Universal Robots PolyScope program: palety_venclovsky.urp

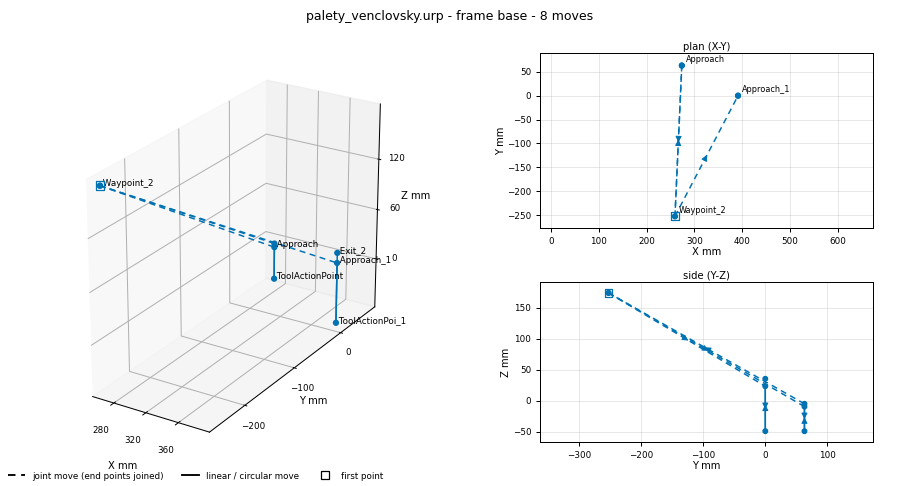
[picture p0: tool path of palety_venclovsky.urp in frame base, 8 of 8 moves have a stored position in this frame; points joined in program order, loops and branches not executed]
Program palety_venclovsky (installation=default directory=/programs/usbdisk createdIn=5.21.2 lastSavedIn=5.21.2 robotSerialNumber=20185300578)
Calibrated DH parameters: a=[-0.000189, -0.243548, -0.212949, 0.000139, -0.000171, 0]; d=[0.151928, 2.340352, -3.79233, 1.582506, 0.085299, 0.092103]; alpha=[1.570802, 0.003282, -0.008312, 1.570809, -1.571939, 0]; deltaTheta=[0, 0.031526, 6.30827, -0.05661, 0, 0]
InitVariablesNode variables(variable(name=Pallet_1_cnt, expression=1), variable(name=Pallet_1_lct, expression=1), variable(name=Pallet_1_lno, expression=1), variable(name=Pallet_1_sep, expression=False), variable(name=Pallet_1_tct, expression=1), variable(name=Pallet_2_cnt, expression=1), variable(name=Pallet_2_lct, expression=1), variable(name=Pallet_2_lno, expression=1), variable(name=Pallet_2_sep, expression=False), variable(name=Pallet_2_tct, expression=1), variable(name=qNearApproach, expression=[0,0,0,0,0,0]), variable(name=qNearApproach_1, expression=[0,0,0,0,0,0]))
BeforeStart
  pocitadlo := 0
  URCap Gripper Activate (Robotiq_Grippers, Robotiq Inc.) dataModel(ResetAndActivateKey=false)
Robot Program (runOnlyOnce=false)
  Call pas_on
  Wait DigitalInput pin=digital_in[2]; digitalValue=1
  URCap Gripper (Robotiq_Grippers, Robotiq Inc.) dataModel(position=100.0, force=54.0, speed=70.0, positionInDouble=100.0, forceInDouble=54.0, speedInDouble=70.0, slaveIds=[9], blocking=true, robotCompliant=false)
  MoveJ speed 60 deg/s, acceleration 80 deg/s^2 (useActiveTCP=true optimoveEnabled=false optiMoveSpeed=0.3 optiMoveAcceleration=0.09) feature=Base
    Waypoint Waypoint_2: TCP in base x=259.302 y=-252.628 z=173.963 mm, rx=-2.2194 ry=2.2233 rz=0.0001 rad; joints [-23.019, -99.618, -73.74, -96.577, 89.565, -23.023] deg; TCP offset x=0 y=0 z=150 mm, rx=0 ry=0 rz=0 rad
  Call pas_off
  If pocitadlo<6
    MoveL speed 180 mm/s, acceleration 1200 mm/s^2 (useActiveTCP=true optimoveEnabled=false optiMoveSpeed=0.3 optiMoveAcceleration=0.09) feature=Base
      MoveDirectionNode (selectedDirection=ZMinus)
        Until TOOL_CONTACT_DETECTION (allowActions=true retraction=0.005 decelerationAcceleration=3 decelerationAngularAcceleration=34.906585)
          MoveDirectionNode (selectedDirection=ZPlus)
            Until DISTANCE (allowActions=false deceleration=3 distanceNodeType=STOP) Distance=0.01; motionParameters(blendRadius=0)
          URCap Gripper (Robotiq_Grippers, Robotiq Inc.) dataModel(position=0.0, force=1.1764705882352942, speed=80.0, positionInDouble=0.0, forceInDouble=1.1764705882352942, speedInDouble=80.0, slaveIds=[9], blocking=true, robotCompliant=false)
          MoveDirectionNode (selectedDirection=ZMinus)
            Until DISTANCE (allowActions=false deceleration=3 distanceNodeType=STOP) Distance=0.025; motionParameters(blendRadius=0)
          pocitadlo := pocitadlo+1
          URCap Gripper (Robotiq_Grippers, Robotiq Inc.) dataModel(position=44.31372549019608, force=39.0, speed=70.0, positionInDouble=44.31372549019608, forceInDouble=39.0, speedInDouble=70.0, slaveIds=[9], blocking=true, robotCompliant=false)
          MoveDirectionNode (selectedDirection=ZPlus)
            Until DISTANCE (allowActions=false deceleration=3 distanceNodeType=STOP) Distance=0.06; motionParameters(blendRadius=0)
          Call pas_off
          URCap Palletizing (polyscope-pallet-impl, Universal Robots) dataModel(palletFeature=Base, isPalletizing=true, rememberTraversal=false, Length(key=objectHeight value=0.03 unit=M), Variable(key=referencePoint, variable(featureName=referencePoint)), Variable(key=separatorPoint, variable(featureName=separatorPoint)), Variable(key=qNearApproach, variable(name=qNearApproach, initializeExpression=[0,0,0,0,0,0])), Variable(key=layerCountingVariable, variable(name=Pallet_1_lct, initializeExpression=1)), Variable(key=layerNumberVariable, variable(name=Pallet_1_lno, initializeExpression=1)), Variable(key=handleSeparatorVariable, variable(name=Pallet_1_sep, initializeExpression=False)), Variable(key=totalCountVariable, variable(name=Pallet_1_tct, initializeExpression=1)), Variable(key=name, variable(name=Pallet_1)), Variable(key=globalCountingVariable, variable(name=Pallet_1_cnt, initializeExpression=1))); state(isChildrenLocked=true)
            URCap Patterns (polyscope-pallet-impl, Universal Robots) state(isChildrenLocked=true)
              URCap Pattern (polyscope-pallet-impl, Universal Robots) dataModel(UUID=a1afcf7f-e893-493d-b622-6c9d734d3802, patternType=GRID, rows=3, columns=2, Variable(key=nameVariable, variable(name=Grid_Pattern_1))); state(isChildrenLocked=true)
                URCap Item (polyscope-pallet-impl, Universal Robots) dataModel(UUID=0f84a695-5284-41e9-b3d2-203e22c0e9f4, patternType=GRID, index=0, calibrationDeltaTheta=[-9.679944364821003E-8, 0.03152637960071048, 6.308270136326222, -0.05660981424064361, 2.1302738175549285E-7, -3.4337321612454286E-7], calibrationA=[-1.89170984734602E-4, -0.24354794633452972, -0.2129485167088614, 1.3892904611349137E-4, -1.7067015336856014E-4, 0.0], calibrationD=[0.15192760230984942, 2.3403518756598336, -3.792330157129607, 1.5825055280731988, 0.08529876240250026, 0.09210299655971649], calibrationAlpha=[1.5708023866418512, 0.0032819461853986743, -0.008311935193061136, 1.570808769909054, -1.5719389687286305, 0.0], calibrationJointChecksum=[-1323472732, -1322302140, 655890344, -1781272900, -1781497016, -1329631202], calibrationStatus=2, calibrationValidChecksum=true, baseToFeature=[0.0, 0.0, 0.0, 0.0, 0.0, 0.0], TCPOffset=[3.46987351703687E-4, -7.600627802391707E-4, 0.2251579720144376, 1.768906187287919E-5, 2.956695373762668E-5, -0.002830388265502223], JointPositions(key=jointpositions, JointPosition(key=[1], Angle(key=pos value=0.712932 unit=RAD)), JointPosition(key=[2], Angle(key=pos value=-1.536445 unit=RAD)), JointPosition(key=[3], Angle(key=pos value=-2.239352 unit=RAD)), JointPosition(key=[4], Angle(key=pos value=-0.935455 unit=RAD)), JointPosition(key=[5], Angle(key=pos value=1.563636 unit=RAD)), JointPosition(key=[6], Angle(key=pos value=-0.86287 unit=RAD))), Variable(key=variable, variable(name=CornerItem_1)))
                URCap Item (polyscope-pallet-impl, Universal Robots) dataModel(UUID=4917496b-efcc-468c-8b87-0b4eec043f87, patternType=GRID, index=1, calibrationDeltaTheta=[-9.679944364821003E-8, 0.03152637960071048, 6.308270136326222, -0.05660981424064361, 2.1302738175549285E-7, -3.4337321612454286E-7], calibrationA=[-1.89170984734602E-4, -0.24354794633452972, -0.2129485167088614, 1.3892904611349137E-4, -1.7067015336856014E-4, 0.0], calibrationD=[0.15192760230984942, 2.3403518756598336, -3.792330157129607, 1.5825055280731988, 0.08529876240250026, 0.09210299655971649], calibrationAlpha=[1.5708023866418512, 0.0032819461853986743, -0.008311935193061136, 1.570808769909054, -1.5719389687286305, 0.0], calibrationJointChecksum=[-1323472732, -1322302140, 655890344, -1781272900, -1781497016, -1329631202], calibrationStatus=2, calibrationValidChecksum=true, baseToFeature=[0.0, 0.0, 0.0, 0.0, 0.0, 0.0], TCPOffset=[3.3288055820729356E-4, -7.179712004344516E-4, 0.22518613724958014, -6.51308584616644E-5, -5.815327347860047E-5, -0.0026860162808949157], JointPositions(key=jointpositions, JointPosition(key=[1], Angle(key=pos value=0.493777 unit=RAD)), JointPosition(key=[2], Angle(key=pos value=-2.007679 unit=RAD)), JointPosition(key=[3], Angle(key=pos value=-1.645848 unit=RAD)), JointPosition(key=[4], Angle(key=pos value=-1.057707 unit=RAD)), JointPosition(key=[5], Angle(key=pos value=1.564628 unit=RAD)), JointPosition(key=[6], Angle(key=pos value=-1.087185 unit=RAD))), Variable(key=variable, variable(name=CornerItem_2)))
                URCap Item (polyscope-pallet-impl, Universal Robots) dataModel(UUID=17d65b1d-739d-439a-9630-1cad21d49f15, patternType=GRID, index=2, calibrationDeltaTheta=[-9.679944364821003E-8, 0.03152637960071048, 6.308270136326222, -0.05660981424064361, 2.1302738175549285E-7, -3.4337321612454286E-7], calibrationA=[-1.89170984734602E-4, -0.24354794633452972, -0.2129485167088614, 1.3892904611349137E-4, -1.7067015336856014E-4, 0.0], calibrationD=[0.15192760230984942, 2.3403518756598336, -3.792330157129607, 1.5825055280731988, 0.08529876240250026, 0.09210299655971649], calibrationAlpha=[1.5708023866418512, 0.0032819461853986743, -0.008311935193061136, 1.570808769909054, -1.5719389687286305, 0.0], calibrationJointChecksum=[-1323472732, -1322302140, 655890344, -1781272900, -1781497016, -1329631202], calibrationStatus=2, calibrationValidChecksum=true, baseToFeature=[0.0, 0.0, 0.0, 0.0, 0.0, 0.0], TCPOffset=[3.5344163164441333E-4, -7.52499091124919E-4, 0.2251565599680179, 4.465585933927923E-6, 3.067966499632582E-5, -0.0027840861433366514], JointPositions(key=jointpositions, JointPosition(key=[1], Angle(key=pos value=0.3406 unit=RAD)), JointPosition(key=[2], Angle(key=pos value=-1.990637 unit=RAD)), JointPosition(key=[3], Angle(key=pos value=-1.675639 unit=RAD)), JointPosition(key=[4], Angle(key=pos value=-1.044914 unit=RAD)), JointPosition(key=[5], Angle(key=pos value=1.564624 unit=RAD)), JointPosition(key=[6], Angle(key=pos value=-1.242929 unit=RAD))), Variable(key=variable, variable(name=CornerItem_3)))
                URCap Item (polyscope-pallet-impl, Universal Robots) dataModel(UUID=e23a75e9-c512-4699-9fb0-38c1f641661b, patternType=GRID, index=3, calibrationDeltaTheta=[-9.679944364821003E-8, 0.03152637960071048, 6.308270136326222, -0.05660981424064361, 2.1302738175549285E-7, -3.4337321612454286E-7], calibrationA=[-1.89170984734602E-4, -0.24354794633452972, -0.2129485167088614, 1.3892904611349137E-4, -1.7067015336856014E-4, 0.0], calibrationD=[0.15192760230984942, 2.3403518756598336, -3.792330157129607, 1.5825055280731988, 0.08529876240250026, 0.09210299655971649], calibrationAlpha=[1.5708023866418512, 0.0032819461853986743, -0.008311935193061136, 1.570808769909054, -1.5719389687286305, 0.0], calibrationJointChecksum=[-1323472732, -1322302140, 655890344, -1781272900, -1781497016, -1329631202], calibrationStatus=2, calibrationValidChecksum=true, baseToFeature=[0.0, 0.0, 0.0, 0.0, 0.0, 0.0], TCPOffset=[3.5491326159248215E-4, -7.352154795082138E-4, 0.22516187238070134, -5.903850028089745E-5, 3.090088451041777E-5, -0.0028011796468691915], JointPositions(key=jointpositions, JointPosition(key=[1], Angle(key=pos value=0.501609 unit=RAD)), JointPosition(key=[2], Angle(key=pos value=-1.50856 unit=RAD)), JointPosition(key=[3], Angle(key=pos value=-2.27851 unit=RAD)), JointPosition(key=[4], Angle(key=pos value=-0.924139 unit=RAD)), JointPosition(key=[5], Angle(key=pos value=1.563638 unit=RAD)), JointPosition(key=[6], Angle(key=pos value=-1.073597 unit=RAD))), Variable(key=variable, variable(name=CornerItem_4)))
            URCap Layers (polyscope-pallet-impl, Universal Robots) dataModel(selectedPatterns=[a1afcf7f-e893-493d-b622-6c9d734d3802], separators=[false])
            URCap At Each Item (polyscope-pallet-impl, Universal Robots) dataModel(selectedPattern=a1afcf7f-e893-493d-b622-6c9d734d3802, selectedPosition=0f84a695-5284-41e9-b3d2-203e22c0e9f4, Approach_calibrationDeltaTheta=[-9.679944364821003E-8, 0.03152637960071048, 6.308270136326222, -0.05660981424064361, 2.1302738175549285E-7, -3.4337321612454286E-7], Approach_calibrationA=[-1.89170984734602E-4, -0.24354794633452972, -0.2129485167088614, 1.3892904611349137E-4, -1.7067015336856014E-4, 0.0], Approach_calibrationD=[0.15192760230984942, 2.3403518756598336, -3.792330157129607, 1.5825055280731988, 0.08529876240250026, 0.09210299655971649], Approach_calibrationAlpha=[1.5708023866418512, 0.0032819461853986743, -0.008311935193061136, 1.570808769909054, -1.5719389687286305, 0.0], Approach_calibrationJointChecksum=[-1323472732, -1322302140, 655890344, -1781272900, -1781497016, -1329631202], Approach_calibrationStatus=2, Approach_calibrationValidChecksum=true, Approach_baseToFeature=[0.0, 0.0, 0.0, 0.0, 0.0, 0.0], Approach_TCPOffset=[3.426090968767226E-4, -7.410222825070811E-4, 0.2251722220319323, -3.696212188149479E-5, -1.49889783493022E-5, -0.0027893122367816064], Exit_calibrationDeltaTheta=[-9.679944364821003E-8, 0.03152637960071048, 6.308270136326222, -0.05660981424064361, 2.1302738175549285E-7, -3.4337321612454286E-7], Exit_calibrationA=[-1.89170984734602E-4, -0.24354794633452972, -0.2129485167088614, 1.3892904611349137E-4, -1.7067015336856014E-4, 0.0], Exit_calibrationD=[0.15192760230984942, 2.3403518756598336, -3.792330157129607, 1.5825055280731988, 0.08529876240250026, 0.09210299655971649], Exit_calibrationAlpha=[1.5708023866418512, 0.0032819461853986743, -0.008311935193061136, 1.570808769909054, -1.5719389687286305, 0.0], Exit_calibrationJointChecksum=[-1323472732, -1322302140, 655890344, -1781272900, -1781497016, -1329631202], Exit_calibrationStatus=2, Exit_calibrationValidChecksum=true, Exit_baseToFeature=[0.0, 0.0, 0.0, 0.0, 0.0, 0.0], Exit_TCPOffset=[3.534060554490903E-4, -7.328819302233058E-4, 0.22516274782089438, -5.956694931654154E-5, 2.1349790715159343E-5, -0.0027647185049195196], currentWizardState=LANDING, Pose(key=refBaseToFeature, Position(key=posePosition, Length(key=X value=0 unit=M), Length(key=Y value=0 unit=M), Length(key=Z value=0 unit=M)), Rotation(key=poseRotation, Angle(key=RX value=0 unit=RAD), Angle(key=RY value=0 unit=RAD), Angle(key=RZ value=0 unit=RAD))), Pose(key=refPose, Position(key=posePosition, Length(key=X value=0.273602 unit=M), Length(key=Y value=0.063177 unit=M), Length(key=Z value=-0.048894 unit=M)), Rotation(key=poseRotation, Angle(key=RX value=-3.14157 unit=RAD), Angle(key=RY value=-0.000044 unit=RAD), Angle(key=RZ value=0.000006 unit=RAD))), JointPositions(key=Approach_jointpositions, JointPosition(key=[1], Angle(key=pos value=0.712584 unit=RAD)), JointPosition(key=[2], Angle(key=pos value=-1.43678 unit=RAD)), JointPosition(key=[3], Angle(key=pos value=-2.112351 unit=RAD)), JointPosition(key=[4], Angle(key=pos value=-1.162056 unit=RAD)), JointPosition(key=[5], Angle(key=pos value=1.562491 unit=RAD)), JointPosition(key=[6], Angle(key=pos value=-0.861559 unit=RAD))), JointPositions(key=Exit_jointpositions, JointPosition(key=[1], Angle(key=pos value=0.712541 unit=RAD)), JointPosition(key=[2], Angle(key=pos value=-1.42836 unit=RAD)), JointPosition(key=[3], Angle(key=pos value=-2.096272 unit=RAD)), JointPosition(key=[4], Angle(key=pos value=-1.186556 unit=RAD)), JointPosition(key=[5], Angle(key=pos value=1.562396 unit=RAD)), JointPosition(key=[6], Angle(key=pos value=-0.861405 unit=RAD))))
              URCap Generated Movements (polyscope-pallet-impl, Universal Robots) state(isChildrenLocked=true)
                MoveJ speed 60 deg/s, acceleration 80 deg/s^2 (useActiveTCP=true optimoveEnabled=false optiMoveSpeed=0.3 optiMoveAcceleration=0.09) feature=referencePoint
                  Waypoint Approach: TCP in base x=273.604 y=63.18 z=-9.252 mm, rx=-3.1416 ry=-0.0001 rz=0 rad; joints [40.828, -82.321, -121.029, -66.581, 89.524, -49.364] deg; TCP offset x=0.343 y=-0.741 z=225.172 mm, rx=0 ry=0 rz=-0.0028 rad; feature pose in base x=273.602 y=63.177 z=-48.894 mm, rx=-3.1416 ry=0 rz=0 rad
                MoveL speed 250 mm/s, acceleration 1200 mm/s^2 (useActiveTCP=true optimoveEnabled=false optiMoveSpeed=0.3 optiMoveAcceleration=0.09) feature(featureName=referencePoint)
                  Waypoint ToolActionPoint: TCP in base x=273.602 y=63.176 z=-48.894 mm, rx=-3.1416 ry=0 rz=0 rad; joints [40.848, -88.032, -128.305, -53.598, 89.59, -49.439] deg; TCP offset x=0.347 y=-0.76 z=225.158 mm, rx=0 ry=0 rz=-0.0028 rad
                Folder Tool action
                  URCap Gripper (Robotiq_Grippers, Robotiq Inc.) dataModel(position=0.0, force=1.1764705882352942, speed=0.0, positionInDouble=0.0, forceInDouble=1.1764705882352942, speedInDouble=0.0, slaveIds=[9], blocking=true, robotCompliant=false)
                MoveL speed 250 mm/s, acceleration 1200 mm/s^2 (useActiveTCP=true optimoveEnabled=false optiMoveSpeed=0.3 optiMoveAcceleration=0.09) feature(featureName=referencePoint)
                  Waypoint Exit_1: TCP in base x=273.614 y=63.172 z=-4.715 mm, rx=-3.1416 ry=0 rz=0 rad; joints [40.826, -81.839, -120.108, -67.985, 89.519, -49.355] deg; TCP offset x=0.353 y=-0.733 z=225.163 mm, rx=-0.0001 ry=0 rz=-0.0028 rad
          MoveJ speed 60 deg/s, acceleration 80 deg/s^2 (useActiveTCP=true optimoveEnabled=false optiMoveSpeed=0.3 optiMoveAcceleration=0.09) feature=Base
            Waypoint Waypoint_2: TCP in base x=259.302 y=-252.628 z=173.963 mm, rx=-2.2194 ry=2.2233 rz=0.0001 rad; joints [-23.019, -99.618, -73.74, -96.577, 89.565, -23.023] deg; TCP offset x=0 y=0 z=150 mm, rx=0 ry=0 rz=0 rad
  If pocitadlo≥6 and pocitadlo<13
    pocitadlo := pocitadlo+1
    URCap Palletizing (polyscope-pallet-impl, Universal Robots) dataModel(palletFeature=Base, isPalletizing=false, Length(key=objectHeight value=0.03 unit=M), Variable(key=referencePoint, variable(featureName=referencePoin_1)), Variable(key=separatorPoint, variable(featureName=separatorPoin_1)), Variable(key=qNearApproach, variable(name=qNearApproach_1, initializeExpression=[0,0,0,0,0,0])), Variable(key=name, variable(name=Pallet_2)), Variable(key=globalCountingVariable, variable(name=Pallet_2_cnt, initializeExpression=1)), Variable(key=layerCountingVariable, variable(name=Pallet_2_lct, initializeExpression=1)), Variable(key=layerNumberVariable, variable(name=Pallet_2_lno, initializeExpression=1)), Variable(key=handleSeparatorVariable, variable(name=Pallet_2_sep, initializeExpression=False)), Variable(key=totalCountVariable, variable(name=Pallet_2_tct, initializeExpression=1))); state(isChildrenLocked=true)
      URCap Patterns (polyscope-pallet-impl, Universal Robots) state(isChildrenLocked=true)
        URCap Pattern (polyscope-pallet-impl, Universal Robots) dataModel(UUID=803d7922-a80b-4571-a540-a1ba350e044b, patternType=GRID, rows=4, columns=3, Variable(key=nameVariable, variable(name=Grid_Pattern_2))); state(isChildrenLocked=true)
          URCap Item (polyscope-pallet-impl, Universal Robots) dataModel(UUID=268bf993-29d4-4b25-8e5d-7caee91635a5, patternType=GRID, index=0, calibrationDeltaTheta=[-9.679944364821003E-8, 0.03152637960071048, 6.308270136326222, -0.05660981424064361, 2.1302738175549285E-7, -3.4337321612454286E-7], calibrationA=[-1.89170984734602E-4, -0.24354794633452972, -0.2129485167088614, 1.3892904611349137E-4, -1.7067015336856014E-4, 0.0], calibrationD=[0.15192760230984942, 2.3403518756598336, -3.792330157129607, 1.5825055280731988, 0.08529876240250026, 0.09210299655971649], calibrationAlpha=[1.5708023866418512, 0.0032819461853986743, -0.008311935193061136, 1.570808769909054, -1.5719389687286305, 0.0], calibrationJointChecksum=[-1323472732, -1322302140, 655890344, -1781272900, -1781497016, -1329631202], calibrationStatus=2, calibrationValidChecksum=true, baseToFeature=[0.0, 0.0, 0.0, 0.0, 0.0, 0.0], TCPOffset=[3.661787772014091E-4, -7.42815896043662E-4, 0.22512024010796766, 5.238855540623789E-6, 1.2098691058805812E-4, -0.002754316056716514], JointPositions(key=jointpositions, JointPosition(key=[1], Angle(key=pos value=0.341525 unit=RAD)), JointPosition(key=[2], Angle(key=pos value=-1.987897 unit=RAD)), JointPosition(key=[3], Angle(key=pos value=-1.672515 unit=RAD)), JointPosition(key=[4], Angle(key=pos value=-1.050806 unit=RAD)), JointPosition(key=[5], Angle(key=pos value=1.564621 unit=RAD)), JointPosition(key=[6], Angle(key=pos value=-1.207811 unit=RAD))), Variable(key=variable, variable(name=CornerItem_5)))
          URCap Item (polyscope-pallet-impl, Universal Robots) dataModel(UUID=fbfc3ace-ba43-4c66-b2fc-4f574954b994, patternType=GRID, index=1, calibrationDeltaTheta=[-9.679944364821003E-8, 0.03152637960071048, 6.308270136326222, -0.05660981424064361, 2.1302738175549285E-7, -3.4337321612454286E-7], calibrationA=[-1.89170984734602E-4, -0.24354794633452972, -0.2129485167088614, 1.3892904611349137E-4, -1.7067015336856014E-4, 0.0], calibrationD=[0.15192760230984942, 2.3403518756598336, -3.792330157129607, 1.5825055280731988, 0.08529876240250026, 0.09210299655971649], calibrationAlpha=[1.5708023866418512, 0.0032819461853986743, -0.008311935193061136, 1.570808769909054, -1.5719389687286305, 0.0], calibrationJointChecksum=[-1323472732, -1322302140, 655890344, -1781272900, -1781497016, -1329631202], calibrationStatus=2, calibrationValidChecksum=true, baseToFeature=[0.0, 0.0, 0.0, 0.0, 0.0, 0.0], TCPOffset=[3.3235696105243795E-4, -7.37485159413024E-4, 0.2251724267316266, -3.0114950725307417E-5, -4.0429256951625296E-5, -0.0027579758966432143], JointPositions(key=jointpositions, JointPosition(key=[1], Angle(key=pos value=0.511316 unit=RAD)), JointPosition(key=[2], Angle(key=pos value=-1.500199 unit=RAD)), JointPosition(key=[3], Angle(key=pos value=-2.272635 unit=RAD)), JointPosition(key=[4], Angle(key=pos value=-0.938231 unit=RAD)), JointPosition(key=[5], Angle(key=pos value=1.563487 unit=RAD)), JointPosition(key=[6], Angle(key=pos value=-1.039039 unit=RAD))), Variable(key=variable, variable(name=CornerItem_6)))
          URCap Item (polyscope-pallet-impl, Universal Robots) dataModel(UUID=ba28164a-2bbb-47bb-8401-54278c357c69, patternType=GRID, index=2, calibrationDeltaTheta=[-9.679944364821003E-8, 0.03152637960071048, 6.308270136326222, -0.05660981424064361, 2.1302738175549285E-7, -3.4337321612454286E-7], calibrationA=[-1.89170984734602E-4, -0.24354794633452972, -0.2129485167088614, 1.3892904611349137E-4, -1.7067015336856014E-4, 0.0], calibrationD=[0.15192760230984942, 2.3403518756598336, -3.792330157129607, 1.5825055280731988, 0.08529876240250026, 0.09210299655971649], calibrationAlpha=[1.5708023866418512, 0.0032819461853986743, -0.008311935193061136, 1.570808769909054, -1.5719389687286305, 0.0], calibrationJointChecksum=[-1323472732, -1322302140, 655890344, -1781272900, -1781497016, -1329631202], calibrationStatus=2, calibrationValidChecksum=true, baseToFeature=[0.0, 0.0, 0.0, 0.0, 0.0, 0.0], TCPOffset=[3.621650591404957E-4, -7.471040884697647E-4, 0.2251650042961146, -4.5052800951793355E-5, 3.650048036724864E-5, -0.0027688463949769506], JointPositions(key=jointpositions, JointPosition(key=[1], Angle(key=pos value=0.709001 unit=RAD)), JointPosition(key=[2], Angle(key=pos value=-1.535335 unit=RAD)), JointPosition(key=[3], Angle(key=pos value=-2.240231 unit=RAD)), JointPosition(key=[4], Angle(key=pos value=-0.935463 unit=RAD)), JointPosition(key=[5], Angle(key=pos value=1.563583 unit=RAD)), JointPosition(key=[6], Angle(key=pos value=-0.878404 unit=RAD))), Variable(key=variable, variable(name=CornerItem_7)))
          URCap Item (polyscope-pallet-impl, Universal Robots) dataModel(UUID=6f5e8f68-d992-4b1d-8750-90dfb2af35b5, patternType=GRID, index=3, calibrationDeltaTheta=[-9.679944364821003E-8, 0.03152637960071048, 6.308270136326222, -0.05660981424064361, 2.1302738175549285E-7, -3.4337321612454286E-7], calibrationA=[-1.89170984734602E-4, -0.24354794633452972, -0.2129485167088614, 1.3892904611349137E-4, -1.7067015336856014E-4, 0.0], calibrationD=[0.15192760230984942, 2.3403518756598336, -3.792330157129607, 1.5825055280731988, 0.08529876240250026, 0.09210299655971649], calibrationAlpha=[1.5708023866418512, 0.0032819461853986743, -0.008311935193061136, 1.570808769909054, -1.5719389687286305, 0.0], calibrationJointChecksum=[-1323472732, -1322302140, 655890344, -1781272900, -1781497016, -1329631202], calibrationStatus=2, calibrationValidChecksum=true, baseToFeature=[0.0, 0.0, 0.0, 0.0, 0.0, 0.0], TCPOffset=[3.406200229312817E-4, -7.20698301989918E-4, 0.22517598600270367, -9.487689101711734E-5, -7.735827791984718E-6, -0.002778372816161836], JointPositions(key=jointpositions, JointPosition(key=[1], Angle(key=pos value=0.498383 unit=RAD)), JointPosition(key=[2], Angle(key=pos value=-2.003753 unit=RAD)), JointPosition(key=[3], Angle(key=pos value=-1.64777 unit=RAD)), JointPosition(key=[4], Angle(key=pos value=-1.059477 unit=RAD)), JointPosition(key=[5], Angle(key=pos value=1.564597 unit=RAD)), JointPosition(key=[6], Angle(key=pos value=-1.087866 unit=RAD))), Variable(key=variable, variable(name=CornerItem_8)))
      URCap Layers (polyscope-pallet-impl, Universal Robots) dataModel(separators=[false], selectedPatterns=[803d7922-a80b-4571-a540-a1ba350e044b])
      URCap At Each Item (polyscope-pallet-impl, Universal Robots) dataModel(selectedPattern=803d7922-a80b-4571-a540-a1ba350e044b, selectedPosition=268bf993-29d4-4b25-8e5d-7caee91635a5, Approach_calibrationDeltaTheta=[-9.679944364821003E-8, 0.03152637960071048, 6.308270136326222, -0.05660981424064361, 2.1302738175549285E-7, -3.4337321612454286E-7], Approach_calibrationA=[-1.89170984734602E-4, -0.24354794633452972, -0.2129485167088614, 1.3892904611349137E-4, -1.7067015336856014E-4, 0.0], Approach_calibrationD=[0.15192760230984942, 2.3403518756598336, -3.792330157129607, 1.5825055280731988, 0.08529876240250026, 0.09210299655971649], Approach_calibrationAlpha=[1.5708023866418512, 0.0032819461853986743, -0.008311935193061136, 1.570808769909054, -1.5719389687286305, 0.0], Approach_calibrationJointChecksum=[-1323472732, -1322302140, 655890344, -1781272900, -1781497016, -1329631202], Approach_calibrationStatus=2, Approach_calibrationValidChecksum=true, Approach_baseToFeature=[0.0, 0.0, 0.0, 0.0, 0.0, 0.0], Approach_TCPOffset=[3.3232136394162337E-4, -6.745512020962623E-4, 0.2251835498426595, -9.63501402427794E-5, -5.0609330485725655E-5, -0.0026252599992773545], Exit_calibrationDeltaTheta=[-9.679944364821003E-8, 0.03152637960071048, 6.308270136326222, -0.05660981424064361, 2.1302738175549285E-7, -3.4337321612454286E-7], Exit_calibrationA=[-1.89170984734602E-4, -0.24354794633452972, -0.2129485167088614, 1.3892904611349137E-4, -1.7067015336856014E-4, 0.0], Exit_calibrationD=[0.15192760230984942, 2.3403518756598336, -3.792330157129607, 1.5825055280731988, 0.08529876240250026, 0.09210299655971649], Exit_calibrationAlpha=[1.5708023866418512, 0.0032819461853986743, -0.008311935193061136, 1.570808769909054, -1.5719389687286305, 0.0], Exit_calibrationJointChecksum=[-1323472732, -1322302140, 655890344, -1781272900, -1781497016, -1329631202], Exit_calibrationStatus=2, Exit_calibrationValidChecksum=true, Exit_baseToFeature=[0.0, 0.0, 0.0, 0.0, 0.0, 0.0], Exit_TCPOffset=[3.498002690335289E-4, -7.199836281285756E-4, 0.22517340344102668, -7.072688683356265E-5, 5.1025465307751155E-6, -0.00274100752749404], currentWizardState=LANDING, Pose(key=refBaseToFeature, Position(key=posePosition, Length(key=X value=0 unit=M), Length(key=Y value=0 unit=M), Length(key=Z value=0 unit=M)), Rotation(key=poseRotation, Angle(key=RX value=0 unit=RAD), Angle(key=RY value=0 unit=RAD), Angle(key=RZ value=0 unit=RAD))), Pose(key=refPose, Position(key=posePosition, Length(key=X value=0.39136 unit=M), Length(key=Y value=0.000068 unit=M), Length(key=Z value=-0.04885 unit=M)), Rotation(key=poseRotation, Angle(key=RX value=-3.141292 unit=RAD), Angle(key=RY value=0.039972 unit=RAD), Angle(key=RZ value=-0.000205 unit=RAD))), JointPositions(key=Approach_jointpositions, JointPosition(key=[1], Angle(key=pos value=0.340972 unit=RAD)), JointPosition(key=[2], Angle(key=pos value=-1.881997 unit=RAD)), JointPosition(key=[3], Angle(key=pos value=-1.459395 unit=RAD)), JointPosition(key=[4], Angle(key=pos value=-1.369691 unit=RAD)), JointPosition(key=[5], Angle(key=pos value=1.563505 unit=RAD)), JointPosition(key=[6], Angle(key=pos value=-1.205941 unit=RAD))), JointPositions(key=Exit_jointpositions, JointPosition(key=[1], Angle(key=pos value=0.340861 unit=RAD)), JointPosition(key=[2], Angle(key=pos value=-1.873287 unit=RAD)), JointPosition(key=[3], Angle(key=pos value=-1.413997 unit=RAD)), JointPosition(key=[4], Angle(key=pos value=-1.423801 unit=RAD)), JointPosition(key=[5], Angle(key=pos value=1.563425 unit=RAD)), JointPosition(key=[6], Angle(key=pos value=-1.205612 unit=RAD))))
        URCap Generated Movements (polyscope-pallet-impl, Universal Robots) state(isChildrenLocked=true)
          MoveJ speed 60 deg/s, acceleration 80 deg/s^2 (useActiveTCP=true optimoveEnabled=false optiMoveSpeed=0.3 optiMoveAcceleration=0.09) feature=referencePoin_1
            Waypoint Approach_1: TCP in base x=391.335 y=-0.001 z=23.567 mm, rx=3.1413 ry=-0.0402 rz=0.0001 rad; joints [19.536, -107.83, -83.617, -78.478, 89.582, -69.095] deg; TCP offset x=0.332 y=-0.675 z=225.184 mm, rx=-0.0001 ry=-0.0001 rz=-0.0026 rad; feature pose in base x=391.36 y=0.068 z=-48.85 mm, rx=-3.1413 ry=0.04 rz=-0.0002 rad
          MoveL speed 250 mm/s, acceleration 1200 mm/s^2 (useActiveTCP=true optimoveEnabled=false optiMoveSpeed=0.3 optiMoveAcceleration=0.09) feature(featureName=referencePoin_1)
            Waypoint ToolActionPoi_1: TCP in base x=391.36 y=0.068 z=-48.85 mm, rx=-3.1413 ry=0.04 rz=-0.0002 rad; joints [19.568, -113.898, -95.828, -60.207, 89.646, -69.202] deg; TCP offset x=0.366 y=-0.743 z=225.12 mm, rx=0 ry=0.0001 rz=-0.0028 rad
          Folder Tool action
            URCap Gripper (Robotiq_Grippers, Robotiq Inc.) dataModel(position=100.0, force=1.1764705882352942, speed=80.0, positionInDouble=100.0, forceInDouble=1.1764705882352942, speedInDouble=80.0, slaveIds=[9], blocking=true, robotCompliant=false)
          MoveL speed 250 mm/s, acceleration 1200 mm/s^2 (useActiveTCP=true optimoveEnabled=false optiMoveSpeed=0.3 optiMoveAcceleration=0.09) feature(featureName=referencePoin_1)
            Waypoint Exit_2: TCP in base x=391.357 y=0.045 z=35.576 mm, rx=-3.1413 ry=0.04 rz=-0.0002 rad; joints [19.53, -107.331, -81.016, -81.578, 89.578, -69.076] deg; TCP offset x=0.35 y=-0.72 z=225.173 mm, rx=-0.0001 ry=0 rz=-0.0027 rad
SubProgram -> pas_on
SubProgram -> pas_off
SubProgram pas_on (keepSynchronizedWithDisk=false)
  Set DigitalOutput pin=digital_out[2]; digitalValue=1
SubProgram pas_off (keepSynchronizedWithDisk=false)
  Set DigitalOutput pin=digital_out[2]; digitalValue=0
